	    // Stop moving second leg, with open valve
	    // 20210506_PRA - Valve normal position changed. Without control signal "#Y9_VijaStop_DesZad" is outside (helix stopped), With control signal "#Y9_VijaStop_DesZad" is inside (helix not stopped)
	    // IF #RightLegIndex=1 OR #RightLegIndex=2 THEN
	    IF #RightLegIndex=0 AND "dbTimers".Num[#i2].TT THEN
	      #Y9_VijaStop_DesZad.AutoON := True;
	    END_IF;
	    // Prepare front position for centring
	    IF "dbDigitalSensors".FOTOCELICA_VIJACENJE_DESNOSPREDAJ.InputF AND NOT #FOTOCELICA_DESNO_SPREDAJ_LATCH THEN
	      #RightLegsArrayIndex[1] := "dbDigitalSensors".FOTOCELICA_VIJACENJE_DESNOSPREDAJ.InputF;  // Reset, ko je vijacenje koncano
	      #FOTOCELICA_DESNO_SPREDAJ_LATCH := True;
	    END_IF;
	    IF #RightLegsArrayIndex[1] AND #InsertNewButtom=0 AND #MoveUPDOWN_DESNOSpredaj THEN
	      #Y11_Centri_DesSpr.AutoON := TRUE;
	    END_IF;
	    // Prepare rear position for centring
	    IF "dbDigitalSensors".FOTOCELICA_VIJACENJE_DESNOZADAJ.InputF AND NOT #FOTOCELICA_DESNO_ZADAJ_LATCH THEN
	      #RightLegsArrayIndex[2] := "dbDigitalSensors".FOTOCELICA_VIJACENJE_DESNOZADAJ.InputF;  // Reset, ko je vijacenje koncano
	      #FOTOCELICA_DESNO_ZADAJ_LATCH := True;
	    END_IF;
	    IF #RightLegsArrayIndex[2] AND #InsertNewButtom=0 AND #MoveUPDOWN_DESNOZadaj THEN
	      #Y10_Centri_DesZad.AutoON := TRUE;
	    END_IF;
	    IF #LeftLegIndex=0 OR #RightLegIndex=0 THEN
	      "dbHMIUser".CurrMachineStep := 'Transport nogic na pozicijo centriranja';
	    END_IF;
	    IF #LeftLegIndex=2 OR #RightLegIndex=2 THEN
	      "dbHMIUser".CurrMachineStep := 'Vstavi dno';
	    END_IF;
	    // **************** END - Stop ZADAJ and centring **************** //  
	    END_REGION CENTRIRANJE
	
	    // *************************************************************************** //  
	    // ************************* BEGIN - Button fastening ************************ // 
	    // *************************************************************************** // 
	    IF ("dbDigitalSensors".INDUKTIVEC_PRAVILNA_VLOZITEV_DNA_1.InputF AND "dbDigitalSensors".INDUKTIVEC_PRAVILNA_VLOZITEV_DNA_2.InputF) AND
	      #LeftLegsArrayIndex[1] AND #LeftLegsArrayIndex[2] AND #RightLegsArrayIndex[1] AND #RightLegsArrayIndex[2]
	      AND (#LeftLegIndex=2 AND #RightLegIndex=2) THEN
	      "dbTimers".Num[#i10].PRE  := #DlyToStartButtomFasten;
	      #ButtomFasting_Activated := True;
	    END_IF;
	    // *************************************************************************** // 
	    // ************************** END - Button fastening ************************* // 
	    // *************************************************************************** // 
	  
	    // *************************************************************************** //  
	    // *************** BEGIN - Start moving UP/DOWN and with helix *************** // 
	    // *************************************************************************** //
	    IF (NOT #RegimeHelix AND ("dbDigitalSensors".START_LEVO_NA_VPENJANJU.OSR OR "dbDigitalSensors".START_DESNO_NA_VPENJANJU.OSR) AND
	      (#InsertNewButtom=0 OR #InsertNewButtom=2))
	      THEN
	      #DetectStartButtom := TRUE;
	      #InsertNewButtom := 0; // Actived centering
	    ELSIF (#RegimeHelix AND (#InsertNewButtom=0 OR #InsertNewButtom=3)) THEN // Buttom removed, new inserted THEN
	      #DetectStartButtom := TRUE;
	      #InsertNewButtom := 0; // Actived centering
	    END_IF;
	
	    "dbTimers".Num[#i10].EE := (#ButtomFasting_Activated AND "dbDigitalSensors".FOTO_ZAVESA_KANAL_1.InputF AND "dbDigitalSensors".FOTO_ZAVESA_KANAL_2.InputF) 
	                               AND
	                               (
	                                #DetectStartButtom
	                               );
	
	    IF #ButtomFasting_Activated AND ("dbTimers".Num[#i10].EE AND "dbTimers".Num[#i10].DN) THEN
	      #Helix_Activated := True;
	    END_IF;    
	    IF #Helix_Activated THEN
	      #Y16_VpenjanjeDna.AutoON := True;
	      #VpenjanjeDnaActived     := True;
	      "dbHMIUser".CurrMachineStep := 'Vpenjanje dna aktivirano';
	    END_IF;
	
	    // V13_VijaLevZad_Dvig, V16_VijaLevSpr_Dvig, V6_VijaDesZad_Dvig, V9_VijaDesSpr_Dvig
	    IF #Helix_Activated THEN
	      IF NOT #MovingUPDOWN_Activated THEN // Timer expired only once
	        "dbTimers".Num[#i1].EE  := True;
	        "dbTimers".Num[#i1].PRE := #DlyToFinishButtonFasten; // 2 s
	        // PRA_20212604 - Activated #Y16_VpenjanjeDna after user press START button, before legs automatically were positioned
	        // #MovingUPDOWN_Activated := ("dbTimers".Num[#i1].EE AND "dbTimers".Num[#i1].DN) AND ("dbDigitalSensors".START_LEVO_NA_VPENJANJU.OSR OR "dbDigitalSensors".START_DESNO_NA_VPENJANJU.OSR);
	        
	        IF "dbTimers".Num[#i1].EE AND "dbTimers".Num[#i1].DN THEN
	          #MovingUPDOWN_Activated := True;
	          "dbTimers".Num[#i1].EE := FALSE;
	          "dbTimers".Num[#i1].DN := FALSE;
	        END_IF;
	      END_IF;
	  
	      IF #MovingUPDOWN_Activated AND ("dbDigitalSensors".INDUKTIVEC_PRAVILNA_VLOZITEV_DNA_1.InputF AND "dbDigitalSensors".INDUKTIVEC_PRAVILNA_VLOZITEV_DNA_2.InputF) THEN
	        "dbHMIUser".CurrMachineStep := 'Vijacenje dna v teku';
	
	        REGION VIJACENJE LEVO SPREDAJ
	        // ***** BEGIN - LEVO SPREDAJ ***** //
	        // Latch present leg
	        IF #LeftLegsArrayIndex[1] AND NOT #MoveUPDOWN_LevoSpredaj THEN
	          "dbTimers".Num[#i1].ACC := 0;
	          "dbTimers".Num[#i1].DN  := FALSE;
	          #MoveUPDOWN_LevoSpredaj := True;
	        END_IF;
	        // Start moving with present leg
	        IF #MoveUPDOWN_LevoSpredaj THEN
	          IF #LeftLegsArrayIndex[1] AND NOT #WaitLevoSpredaj THEN
	            #Y5_VijaLevSpr_Dvig.AutoON   := True;
	            #M2_SPREDAJ_LEVO.AutoON      := True;
	            #M2_SPREDAJ_LEVO.Speed1Out   := True;
	          END_IF;
	
	          IF NOT #WaitLevoSpredaj THEN
	            IF #M2_SPREDAJ_LEVO.AutoON THEN
	              "dbTimers".Num[#i1].EE  := #M2_SPREDAJ_LEVO.AutoON;
	              "dbTimers".Num[#i1].PRE  := #DlyToRotateOpposite; // 3 s
	            END_IF;
	            IF ("dbTimers".Num[#i1].EE AND NOT "dbTimers".Num[#i1].DN) THEN
	              #M2_SPREDAJ_LEVO.DirectionReq := True; // Rotate opposite for proper landing leg to button hole
	            ELSIF ("dbTimers".Num[#i1].EE AND "dbTimers".Num[#i1].DN) THEN // Leg needs to touch button and delay expired
	              #M2_SPREDAJ_LEVO.DirectionReq := False; // Change direction to start helix
	            END_IF;
	
	            // Leg hegix succeeded, wait to reach end cilinder position "DVIG_DOL=1"
	            IF (NOT #M2_SPREDAJ_LEVO.DirectionReq AND "dbTimers".Num[#i1].EE AND "dbTimers".Num[#i1].DN) AND ("IND_VIJAC_LEVO_NAPREJ" OR "dbDigitalSensors".KONCNA_POZICIJA_VIJACENJA_LEVO_NAPREJ.InputF) THEN
	              #M2_SPREDAJ_LEVO.AutoON       := False;
	              "dbTimers".Num[#i1].EE        := False;
	              "dbTimers".Num[#i1].DN        := False;
	              "dbTimers".Num[#i1].ACC       := 0;
	             
	              #WaitLevoSpredaj              := True;
	            END_IF;
	          END_IF;
	
	          // Start moving down after timer expired
	          IF #WaitLevoSpredaj THEN
	            "dbTimers".Num[#i1].EE  := True;
	            "dbTimers".Num[#i1].PRE  := #WaitTimeBeforeMoveDown;
	
	            IF "dbTimers".Num[#i1].EE AND NOT "dbTimers".Num[#i1].DN THEN
	              #Y5_VijaLevSpr_Dvig.AutoON    := True; // Dvig gor, till timer expired
	            END_IF;
	
	            // Wait to reached end position
	            IF "dbDigitalSensors".MESTO_VIJACENJE_LEVO_SPRED_DVIG_DOL.InputF THEN
	              #LeftLegsArrayIndex[1]  := "dbDigitalSensors".FOTOCELICA_VIJACENJE_LEVO_SPREDAJ.InputF; // Check if helix present at the end of moving motor down
	              #WaitLevoSpredaj        := False;
	              #MoveUPDOWN_LevoSpredaj := False;
	              #EndLevoSpredaj := True;
	            END_IF;
	          END_IF;
	        END_IF;
	        // ***** END - LEVO SPREDAJ ***** //
	        END_REGION VIJACENJE LEVO SPREDAJ
	
	        REGION VIJACENJE LEVO ZADAJ
	        // ***** BEGIN - LEVO ZADAJ ***** //
	        // Latch present leg
	        IF #LeftLegsArrayIndex[2] AND NOT #MoveUPDOWN_LevoZadaj THEN
	          "dbTimers".Num[#i2].ACC   := 0;
	          "dbTimers".Num[#i2].DN  := FALSE;
	          #MoveUPDOWN_LevoZadaj := True;
	        END_IF;
	        // Start moving with present leg
	        IF #MoveUPDOWN_LevoZadaj THEN
	          IF #LeftLegsArrayIndex[2] AND NOT #WaitLevoZadaj THEN
	            #Y4_VijaLevZad_Dvig.AutoON   := True;
	            #M1_ZADAJ_LEVO.AutoON      := True;
	            #M1_ZADAJ_LEVO.Speed1Out   := True;
	          END_IF;
	
	          IF NOT #WaitLevoZadaj THEN
	            IF #M1_ZADAJ_LEVO.AutoON THEN
	              "dbTimers".Num[#i2].EE  := #M1_ZADAJ_LEVO.AutoON;
	              "dbTimers".Num[#i2].PRE  := #DlyToRotateOpposite; // 3 s
	            END_IF;
	            IF ("dbTimers".Num[#i2].EE AND NOT "dbTimers".Num[#i2].DN) THEN
	              #M1_ZADAJ_LEVO.DirectionReq := True; // Rotate opposite for proper landing leg to button hole
	            ELSIF("dbTimers".Num[#i2].EE AND "dbTimers".Num[#i2].DN) THEN // Leg needs to touch button and delay expired
	              #M1_ZADAJ_LEVO.DirectionReq := False; // Change direction to start helix
	            END_IF;
	
	            // Leg hegix succeeded, wait to reach end cilinder position "DVIG_DOL=1"
	            IF (NOT #M1_ZADAJ_LEVO.DirectionReq AND "dbTimers".Num[#i2].EE AND "dbTimers".Num[#i2].DN) AND ("IND_VIJAC_LEVO_NAZAJ" OR "dbDigitalSensors".KONCNA_POZICIJA_VIJACENJA_LEVO_NAZAJ.InputF ) THEN
	              #M1_ZADAJ_LEVO.AutoON       := False;
	              "dbTimers".Num[#i2].EE        := False;
	              "dbTimers".Num[#i2].DN        := False;
	              "dbTimers".Num[#i2].ACC       := 0;
	
	              #WaitLevoZadaj              := True;
	            END_IF;
	          END_IF;
	
	          // Start moving down after timer expired
	          IF #WaitLevoZadaj THEN
	            "dbTimers".Num[#i2].EE  := True;
	            "dbTimers".Num[#i2].PRE  := #WaitTimeBeforeMoveDown;
	
	            IF "dbTimers".Num[#i2].EE AND NOT "dbTimers".Num[#i2].DN THEN
	              #Y4_VijaLevZad_Dvig.AutoON    := True; // Dvig gor, till timer expired
	            END_IF;
	
	            // Wait to reached end position
	            IF "dbDigitalSensors".MESTO_VIJACENJE_LEVO_ZAD_DVIG_DOL.InputF THEN
	              #LeftLegsArrayIndex[2] := "dbDigitalSensors".FOTOCELICA_VIJACENJE_LEVO_ZADAJ.InputF; // // Check if helix present at the end of moving motor down
	              #WaitLevoZadaj         := False;
	              #MoveUPDOWN_LevoZadaj  := False;
	              #EndLevoZadaj := True;
	            END_IF;
	          END_IF;
	        END_IF;
	        // ***** END - LEVO ZADAJ ***** //
	        END_REGION VIJACENJE LEVO ZADAJ
	
	        REGION VIJACENJE DESNO SPREDAJ
	        // ***** BEGIN - DESNO SPREDAJ ***** //
	        // Latch present leg
	        IF #RightLegsArrayIndex[1] AND NOT #MoveUPDOWN_DESNOSpredaj THEN
	          "dbTimers".Num[#i3].ACC   := 0;
	          "dbTimers".Num[#i3].DN  := FALSE;
	          #MoveUPDOWN_DESNOSpredaj := True;
	        END_IF;
	        // Start moving with present leg
	        IF #MoveUPDOWN_DESNOSpredaj THEN
	          IF #RightLegsArrayIndex[1] AND NOT #WaitDesnoSpredaj THEN
	            #Y3_VijaDesSpr_Dvig.AutoON   := True;
	            #M2_SPREDAJ_DESNO.AutoON      := True;
	            #M2_SPREDAJ_DESNO.Speed1Out   := True;
	          END_IF;
	
	          IF NOT #WaitDesnoSpredaj THEN
	            IF #M2_SPREDAJ_DESNO.AutoON THEN
	              "dbTimers".Num[#i3].EE  := #M2_SPREDAJ_DESNO.AutoON;
	              "dbTimers".Num[#i3].PRE  := #DlyToRotateOpposite; // 3 s
	            END_IF;
	            IF ("dbTimers".Num[#i3].EE AND NOT "dbTimers".Num[#i3].DN) THEN
	              #M2_SPREDAJ_DESNO.DirectionReq := True; // Rotate opposite for proper landing leg to button hole
	            ELSIF ("dbTimers".Num[#i3].EE AND "dbTimers".Num[#i3].DN) THEN // Leg needs to touch button and delay expir
	              #M2_SPREDAJ_DESNO.DirectionReq := False; // Change direction to start helix
	            END_IF;
	
	            // Leg hegix succeeded, wait to reach end cilinder position "DVIG_DOL=1"
	            IF (NOT #M2_SPREDAJ_DESNO.DirectionReq AND "dbTimers".Num[#i3].EE AND "dbTimers".Num[#i3].DN) AND ("IND_VIJAC_DES_NAPREJ" OR "dbDigitalSensors".KONCNA_POZICIJA_VIJACENJA_DES_NAPREJ.InputF) THEN
	              #M2_SPREDAJ_DESNO.AutoON      := False;          
	              "dbTimers".Num[#i3].EE        := False;
	              "dbTimers".Num[#i3].DN        := False;
	              "dbTimers".Num[#i3].ACC       := 0;
	
	              #WaitDesnoSpredaj             := True;
	            END_IF;
	          END_IF;
	
	          // Start moving down after timer expired
	          IF #WaitDesnoSpredaj THEN
	            "dbTimers".Num[#i3].EE  := True;
	            "dbTimers".Num[#i3].PRE  := #WaitTimeBeforeMoveDown;
	
	            IF "dbTimers".Num[#i3].EE AND NOT "dbTimers".Num[#i3].DN THEN
	              #Y3_VijaDesSpr_Dvig.AutoON    := True; // Dvig gor, till timer expired
	            END_IF;
	
	            // Wait to reached end position
	            IF "dbDigitalSensors".MESTO_VIJACENJE_DESNO_SPRED_DVIG_DOL.InputF THEN
	              #RightLegsArrayIndex[1]  := "dbDigitalSensors".FOTOCELICA_VIJACENJE_DESNOSPREDAJ.InputF; // // Check if helix present at the end of moving motor down
	              #WaitDesnoSpredaj        := False;
	              #MoveUPDOWN_DESNOSpredaj := False;
	              #EndDesnoSpredaj := True;
	            END_IF;
	          END_IF;
	        END_IF;
	        // ***** END - DESNO SPREDAJ ***** //
	        END_REGION VIJACENJE DESNO SPREDAJ
	
	        REGION VIJACENJE DESNO ZADAJ
	        // ***** BEGIN - DESNO ZADAJ ***** //
	        // Latch present leg
	        IF #RightLegsArrayIndex[2] AND NOT #MoveUPDOWN_DESNOZadaj THEN
	          "dbTimers".Num[#i4].ACC  := 0;
	          "dbTimers".Num[#i4].DN  := FALSE;
	          #MoveUPDOWN_DESNOZadaj := True;
	        END_IF;
	        // Start moving with present leg
	        IF #MoveUPDOWN_DESNOZadaj THEN
	          IF #RightLegsArrayIndex[2] AND NOT #WaitDesnoZadaj THEN
	            #Y2_VijaDesZad_Dvig.AutoON   := True;
	            #M1_ZADAJ_DESNO.AutoON      := True;
	            #M1_ZADAJ_DESNO.Speed1Out   := True;
	          END_IF;
	
	          IF NOT #WaitDesnoZadaj THEN
	            IF #M1_ZADAJ_DESNO.AutoON THEN
	              "dbTimers".Num[#i4].EE  := #M1_ZADAJ_DESNO.AutoON;
	              "dbTimers".Num[#i4].PRE  := #DlyToRotateOpposite; // 3 s
	            END_IF;
	            IF ("dbTimers".Num[#i4].EE AND NOT "dbTimers".Num[#i4].DN) THEN
	              #M1_ZADAJ_DESNO.DirectionReq := True; // Rotate opposite for proper landing leg to button hole
	            ELSIF ("dbTimers".Num[#i4].EE AND "dbTimers".Num[#i4].DN) THEN // // Leg needs to touch button and delay expired
	              #M1_ZADAJ_DESNO.DirectionReq := False; // Change direction to start helix
	            END_IF;
	
	            // Leg hegix succeeded, wait to reach end cilinder position "DVIG_DOL=1"
	            IF (NOT #M1_ZADAJ_DESNO.DirectionReq AND "dbTimers".Num[#i4].EE AND "dbTimers".Num[#i4].DN) AND ("IND_VIJAC_DES_NAZAJ" OR "dbDigitalSensors".KONCNA_POZICIJA_VIJACENJA_DES_NAZAJ.InputF) THEN 
	              #M1_ZADAJ_DESNO.AutoON       := False;
	              "dbTimers".Num[#i4].EE       := False;
	              "dbTimers".Num[#i4].DN       := False;
	              "dbTimers".Num[#i4].ACC      := 0;
	
	              #WaitDesnoZadaj              := True;
	            END_IF;
	          END_IF;
	
	          // Start moving down after timer expired
	          IF #WaitDesnoZadaj THEN
	            "dbTimers".Num[#i4].EE  := True;
	            "dbTimers".Num[#i4].PRE  := #WaitTimeBeforeMoveDown;
	
	            IF "dbTimers".Num[#i4].EE AND NOT "dbTimers".Num[#i4].DN THEN
	              #Y2_VijaDesZad_Dvig.AutoON    := True; // Dvig gor, till timer expired
	            END_IF;
	
	            // Wait to reached end position
	            IF "dbDigitalSensors".MESTO_VIJACENJE_DESNO_ZAD_DVIG_DOL.InputF THEN
	              #RightLegsArrayIndex[2] := "dbDigitalSensors".FOTOCELICA_VIJACENJE_DESNOZADAJ.InputF; // // Check if helix present at the end of moving motor down
	              #WaitDesnoZadaj        := False;
	              #MoveUPDOWN_DESNOZadaj := False;
	              #EndDesnoZadaj := True;
	            END_IF;
	          END_IF;
	        END_IF;
	        // ***** END - DESNO ZADAJ ***** //
	        END_REGION VIJACENJE DESNO ZADAJ
	
	        // Next step
	        IF (#EndLevoSpredaj AND #EndLevoZadaj AND #EndDesnoSpredaj AND #EndDesnoZadaj) AND
	           ("dbDigitalSensors".FOTO_ZAVESA_KANAL_1.InputF AND "dbDigitalSensors".FOTO_ZAVESA_KANAL_2.InputF)     
	          THEN
	          "dbTimers".Num[#i1].EE  := False;
	          "dbTimers".Num[#i1].DN  := False;
	          "dbTimers".Num[#i1].ACC := 0;
	          "dbTimers".Num[#i2].EE  := False;
	          "dbTimers".Num[#i2].DN  := False;
	          "dbTimers".Num[#i2].ACC := 0;
	          "dbTimers".Num[#i3].EE  := False;
	          "dbTimers".Num[#i3].DN  := False;
	          "dbTimers".Num[#i3].ACC := 0;
	          "dbTimers".Num[#i4].EE  := False;
	          "dbTimers".Num[#i4].DN  := False;
	          "dbTimers".Num[#i4].ACC := 0;
	          "dbTimers".Num[#i10].EE  := False;
	          "dbTimers".Num[#i10].DN  := False;
	          "dbTimers".Num[#i10].ACC := 0;
	          #TotalButtomPlateCounter := #TotalButtomPlateCounter + 1;
	
	          #CurrentStep := 20;
	        END_IF;
	  
	      END_IF; // #MovingUPDOWN_ready
	    END_IF;   // #Helix_Activated
	    // *************************************************************************** // 
	    // *************** END - Start moving UP/DOWN and with helix ***************** //
	    // *************************************************************************** // 
	
	  20:  // Remove button plate - wait user to remove button plate
	  "dbHMIUser".CurrMachineStep := 'Odstrani dno iz naprave';
	  #MovingUPDOWN_Activated := False; // 20210426_PRA Added to reset before plate is removed. Used in fcUtilities->timer: StandbyTimeTrakaVijac
	  #InsertNewButtom := 1;
	
	  IF #LeftLegsArrayIndex[1] OR #LeftLegsArrayIndex[2] THEN
	    #LeftLegIndex  := 2; // vijačenje neuspešno, ponovi vijačenje z istimi nogicami
	  ELSE
	    #LeftLegIndex  := 0; // vijačenje uspešno
	  END_IF;
	  IF #RightLegsArrayIndex[1] OR #RightLegsArrayIndex[2] THEN
	    #RightLegIndex := 2; // vijačenje neuspešno, ponovi vijačenje z istimi nogicami
	  ELSE
	    #RightLegIndex := 0; // vijačenje uspešno
	  END_IF;
	
	  IF #LeftLegIndex=0 AND #RightLegIndex=0 THEN
	    #LegsReadyOnPosToHelix := False;
	  END_IF;
	
	  REGION CENTRIRANJE AT END
	  // *************** BEGIN - Stop ZADAJ and centring *************** //
	  (* // 20210506_PRA In normal position #Y13_VijaStop_LevZad is outside
	  IF #LeftLegIndex=1 OR #LeftLegIndex=2 THEN
	    #Y13_VijaStop_LevZad.AutoON := True;  // Stop moving second leg, with open valve
	  END_IF;
	  *)
	  IF #LeftLegsArrayIndex[1] THEN
	    #Y15_Centri_LevSpr.AutoON := TRUE;
	  END_IF;
	  IF #LeftLegsArrayIndex[2] THEN
	    #Y14_Centri_LevZad.AutoON := TRUE;
	  END_IF;
	
	  (* // 20210506_PRA In normal position #Y9_VijaStop_DesZad is outside
	  IF #RightLegIndex=1 OR #RightLegIndex=2 THEN
	    #Y9_VijaStop_DesZad.AutoON := True; // Stop moving second leg, with open valve
	  END_IF;
	  *)
	  IF #RightLegsArrayIndex[1] THEN
	    #Y11_Centri_DesSpr.AutoON := TRUE;
	  END_IF;
	  IF #RightLegsArrayIndex[2] THEN
	    #Y10_Centri_DesZad.AutoON := TRUE;
	  END_IF;
	  // **************** END - Stop ZADAJ and centring **************** //  
	  END_REGION CENTRIRANJE
	
	  "dbTimers".Num[#i1].FR    := False;
	  "dbTimers".Num[#i2].FR    := False;
	  "dbTimers".Num[#i3].FR    := False;
	  "dbTimers".Num[#i4].FR    := False;
	
	  "dbTimers".Num[#i1].EE := ("dbDigitalSensors".FOTO_ZAVESA_KANAL_1.InputF AND "dbDigitalSensors".FOTO_ZAVESA_KANAL_2.InputF) AND
	                            "dbDigitalSensors".MESTO_VIJACENJE_LEVO_SPRED_DVIG_DOL.InputF AND "dbDigitalSensors".MESTO_VIJACENJE_LEVO_SPRED_DVIG_DOL.InputF AND
	                            "dbDigitalSensors".MESTO_VIJACENJE_DESNO_SPRED_DVIG_DOL.InputF AND "dbDigitalSensors".MESTO_VIJACENJE_DESNO_SPRED_DVIG_DOL.InputF;
	                            // 20210429_PRA Start next legs positions even if buttom was not removed from machine and buttom AND still present
	                            // (NOT "dbDigitalSensors".INDUKTIVEC_PRAVILNA_VLOZITEV_DNA_1.InputF AND NOT "dbDigitalSensors".INDUKTIVEC_PRAVILNA_VLOZITEV_DNA_2.InputF)
	  "dbTimers".Num[#i1].PRE := #WEndTimeToRemovePlate;
	  IF "dbTimers".Num[#i1].EE AND "dbTimers".Num[#i1].DN THEN
	    // *************** BEGIN - Preveri ali so bile nogice zvijacene *************** //
	    #LeftLegsArrayIndex[1] := "dbDigitalSensors".FOTOCELICA_VIJACENJE_LEVO_SPREDAJ.InputF;
	    #LeftLegsArrayIndex[2] := "dbDigitalSensors".FOTOCELICA_VIJACENJE_LEVO_ZADAJ.InputF;
	    #RightLegsArrayIndex[1] := "dbDigitalSensors".FOTOCELICA_VIJACENJE_DESNOSPREDAJ.InputF;
	    #RightLegsArrayIndex[2] := "dbDigitalSensors".FOTOCELICA_VIJACENJE_DESNOZADAJ.InputF;
	    // **************** END - Preveri ali so bile nogice zvijacene **************** //  
	    #CurrentStep := 21;
	  END_IF;
	  
	  21:  // Jump to initial step
	  "dbTimers".Num[#i1].EE  := False;
	  "dbTimers".Num[#i1].DN  := False;
	
	  #InitPosition := False;
	  #CurrentStep := 1; // Check conditions on init step
	
	END_CASE;
	
	// ALARMS SECTION
	  // Alarm 1
	  IF #Y8_VijaLocev_Des.Alarm THEN
	    "dbAlarms".PLI[#PLIIndex, 1] := 1;
	  END_IF;
	  
	  // Alarm 2
	  IF #Y9_VijaStop_DesZad.Alarm THEN
	    "dbAlarms".PLI[#PLIIndex, 2] := 1;
	  END_IF;
	  
	  // Alarm 3
	  IF #Y2_VijaDesZad_Dvig.Alarm THEN
	    "dbAlarms".PLI[#PLIIndex, 3] := 1;
	  END_IF;
	  
	  // Alarm 4
	  IF #Y10_Centri_DesZad.Alarm THEN
	    "dbAlarms".PLI[#PLIIndex, 4] := 1;
	  END_IF;
	  
	  // Alarm 5
	  IF #Y3_VijaDesSpr_Dvig.Alarm THEN
	    "dbAlarms".PLI[#PLIIndex, 5] := 1;
	  END_IF;
	
	  // Alarm 6
	  IF #Y11_Centri_DesSpr.Alarm THEN
	    "dbAlarms".PLI[#PLIIndex, 6] := 1;
	  END_IF;
	
	  // Alarm 7
	  IF #Y12_VijaLocev_Lev.Alarm THEN 
	    "dbAlarms".PLI[#PLIIndex, 7] := 1;
	  END_IF;
	  
	  // Alarm 8
	  IF #Y13_VijaStop_LevZad.Alarm THEN 
	    "dbAlarms".PLI[#PLIIndex, 8] := 1;
	  END_IF;
	  
	  // Alarm 9
	  IF #Y4_VijaLevZad_Dvig.Alarm THEN
	    "dbAlarms".PLI[#PLIIndex, 9] := 1;
	  END_IF;
	  
	  // Alarm 10
	  IF #Y14_Centri_LevZad.Alarm THEN
	    "dbAlarms".PLI[#PLIIndex, 10] := 1;
	  END_IF;
	  
	  // Alarm 11
	  IF #Y5_VijaLevSpr_Dvig.Alarm THEN
	    "dbAlarms".PLI[#PLIIndex, 11] := 1;
	  END_IF;
	  
	  // Alarm 12
	  IF #Y15_Centri_LevSpr.Alarm THEN
	    "dbAlarms".PLI[#PLIIndex, 12] := 1;
	  END_IF;
	
	  // Alarm 13
	  IF #Y16_VpenjanjeDna.Alarm THEN
	    "dbAlarms".PLI[#PLIIndex, 13] := 1;
	  END_IF;
	
	  // Alarm 14
	  IF #M1_ZADAJ_LEVO.Alarm THEN
	    "dbAlarms".PLI[#PLIIndex, 14] := 1;
	  END_IF;
	
	  // Alarm 15
	  IF #M2_SPREDAJ_LEVO.Alarm THEN
	    "dbAlarms".PLI[#PLIIndex, 15] := 1;
	  END_IF;
	
	  // Alarm 16
	  IF #M1_ZADAJ_DESNO.Alarm THEN
	    "dbAlarms".PLI[#PLIIndex, 16] := 1;
	  END_IF;
	
	  // Alarm 17
	  IF #M2_SPREDAJ_DESNO.Alarm THEN
	    "dbAlarms".PLI[#PLIIndex, 17] := 1;
	  END_IF;
	
	  // Alarm 18
	  IF #VKLOP_M_TRAKA_VIJACNIKA.Alarm THEN
	    "dbAlarms".PLI[#PLIIndex, 18] := 1;
	  END_IF;
	
	  // Alarm 19
	  // Začetne pozicije vijačnega dela niso dosežene
	  IF #CurrentStep = 1 AND #IEC_TimerOnDly_DN_1 THEN // NOT #InitPosition
	    "dbAlarms".PLI[#PLIIndex, 19] := 1;
	  END_IF;
	
	  // Alarm 20
	  // Manjka ena od nogic na pozicijah za vijačenje-ročno odstrani nogice
	  IF (#CurrentStep >= 3 AND #CurrentStep <= 5) AND
	    (#LeftLegsArrayIndex[1] XOR #LeftLegsArrayIndex[2] XOR #RightLegsArrayIndex[1] XOR #RightLegsArrayIndex[2])
	  THEN
	    "dbUnit".Unit[1].StartStop := False;
	    "dbAlarms".PLI[#PLIIndex, 20] := 1;
	  END_IF;
	
	  // Alarm 21 - Added 20210512_PRA
	  // Dovoljeni čas vijačenja nogice levo-spredaj potekel
	  "dbTimers".Num[#i5].EE := (#PhaseStatus=5 AND #CurrentStep = 10) AND #MovingUPDOWN_Activated AND #MoveUPDOWN_LevoSpredaj AND NOT #WaitLevoSpredaj;
	  "dbTimers".Num[#i5].PRE := #TimeoutToEndHelix;
	  IF "dbTimers".Num[#i5].EE AND "dbTimers".Num[#i5].DN
	  THEN
	    "dbUnit".Unit[1].StartStop := False;
	    "dbAlarms".PLI[#PLIIndex, 21] := 1;
	  END_IF;
	
	  // Alarm 22 - Added 20210512_PRA
	  // Dovoljeni čas vijačenja nogice levo-zadaj potekel
	  "dbTimers".Num[#i6].EE := (#PhaseStatus=5 AND #CurrentStep = 10) AND #MovingUPDOWN_Activated AND #MoveUPDOWN_LevoZadaj AND NOT #WaitLevoZadaj;
	  "dbTimers".Num[#i6].PRE := #TimeoutToEndHelix;
	  IF "dbTimers".Num[#i6].EE AND "dbTimers".Num[#i6].DN
	  THEN
	    "dbUnit".Unit[1].StartStop := False;
	    "dbAlarms".PLI[#PLIIndex, 22] := 1;
	  END_IF;
	
	  // Alarm 23 - Added 20210512_PRA
	  // Dovoljeni čas vijačenja nogice desno-spredaj potekel
	  "dbTimers".Num[#i7].EE := (#PhaseStatus=5 AND #CurrentStep = 10) AND #MovingUPDOWN_Activated AND #MoveUPDOWN_DESNOSpredaj AND NOT #WaitDesnoSpredaj;
	  "dbTimers".Num[#i7].PRE := #TimeoutToEndHelix;
	  IF "dbTimers".Num[#i7].EE AND "dbTimers".Num[#i7].DN
	  THEN
	    "dbUnit".Unit[1].StartStop := False;
	    "dbAlarms".PLI[#PLIIndex, 23] := 1;
	  END_IF;
	
	  // Alarm 24 - Added 20210512_PRA
	  // Dovoljeni čas vijačenja nogice desno-zadaj potekel
	  "dbTimers".Num[#i8].EE := (#PhaseStatus=5 AND #CurrentStep = 10) AND #MovingUPDOWN_Activated AND #MoveUPDOWN_DESNOZadaj AND NOT #WaitDesnoZadaj;
	  "dbTimers".Num[#i8].PRE := #TimeoutToEndHelix;
	  IF "dbTimers".Num[#i8].EE AND "dbTimers".Num[#i8].DN
	  THEN
	    "dbUnit".Unit[1].StartStop := False;
	    "dbAlarms".PLI[#PLIIndex, 24] := 1;
	  END_IF;
	
	  // Alarms in running state
	  IF #PhaseStatus = 5 THEN
	    IF (NOT #AlarmPresentOLD AND #AlarmPresent) OR (NOT #InitPositionOLD AND #InitPosition) THEN
	      ; // #CurrentStep := 6;
	    END_IF;
	  END_IF;
	
	#AlarmPresentOLD      := #AlarmPresent;
	#InitPositionOLD      := #InitPosition;
	
	IF (#CurrentStep = 10) THEN
	  #LeftLegIndexOLD      := #LeftLegIndex;
	  #RightLegIndexOLD     := #RightLegIndex;
	END_IF;
END_FUNCTION_BLOCK

FUNCTION_BLOCK "ph_LegsShifter_2"
{ S7_Optimized_Access := 'TRUE' }
VERSION : 0.1
   VAR_IN_OUT 
      Y17_RotCilipozDesno : "udtDigitalValve";
      Y18_RotCilipozLevo : "udtDigitalValve";
      Y6_DrcaLocev_Des : "udtDigitalValve";
      Y7_DrcaLocev_Lev : "udtDigitalValve";
   END_VAR

   VAR RETAIN
      CurrentStep { ExternalAccessible := 'False'; ExternalVisible := 'False'; ExternalWritable := 'False'} : Int;
      PhaseStatus { ExternalAccessible := 'False'; ExternalVisible := 'False'; ExternalWritable := 'False'} : Int;   // // 0=IDLE, 5=RUNNING, 6=HOLD
      Mode { ExternalAccessible := 'False'; ExternalVisible := 'False'; ExternalWritable := 'False'} : SInt;
      AlarmPresent { ExternalAccessible := 'False'; ExternalVisible := 'False'; ExternalWritable := 'False'} : Bool;
      InitPosition { ExternalAccessible := 'False'; ExternalVisible := 'False'; ExternalWritable := 'False'} : Bool;
   END_VAR
   VAR 
      StartCmd { ExternalAccessible := 'False'; ExternalVisible := 'False'; ExternalWritable := 'False'} : Bool;
      AlarmPresentOLD { ExternalAccessible := 'False'; ExternalVisible := 'False'; ExternalWritable := 'False'} : Bool;
      InitPositionOLD { ExternalAccessible := 'False'; ExternalVisible := 'False'; ExternalWritable := 'False'} : Bool;
      IEC_TimerOnDly_1 {InstructionName := 'TONR_TIME'; LibVersion := '1.0'; ExternalAccessible := 'False'; ExternalVisible := 'False'; ExternalWritable := 'False'; S7_SetPoint := 'False'} : TONR_TIME;
      IEC_TimerOnDly_2 {InstructionName := 'TONR_TIME'; LibVersion := '1.0'; ExternalAccessible := 'False'; ExternalVisible := 'False'; ExternalWritable := 'False'; S7_SetPoint := 'False'} : TONR_TIME;
      IEC_TimerOnDly_3 {InstructionName := 'TONR_TIME'; LibVersion := '1.0'; ExternalAccessible := 'False'; ExternalVisible := 'False'; ExternalWritable := 'False'; S7_SetPoint := 'False'} : TONR_TIME;
      IEC_TimerOnDly_4 {InstructionName := 'TONR_TIME'; LibVersion := '1.0'; ExternalAccessible := 'False'; ExternalVisible := 'False'; ExternalWritable := 'False'; S7_SetPoint := 'False'} : TONR_TIME;
      IEC_TimerOnDly_5 {InstructionName := 'TONR_TIME'; LibVersion := '1.0'; ExternalAccessible := 'False'; ExternalVisible := 'False'; ExternalWritable := 'False'; S7_SetPoint := 'False'} : TONR_TIME;
      IEC_TimerOnDly_6 {InstructionName := 'TONR_TIME'; LibVersion := '1.0'; ExternalAccessible := 'False'; ExternalVisible := 'False'; ExternalWritable := 'False'; S7_SetPoint := 'False'} : TONR_TIME;
      IEC_TimerOnDly_7 {InstructionName := 'TONR_TIME'; LibVersion := '1.0'; ExternalAccessible := 'False'; ExternalVisible := 'False'; ExternalWritable := 'False'; S7_SetPoint := 'False'} : TONR_TIME;
      IEC_TimerOnDly_8 {InstructionName := 'TONR_TIME'; LibVersion := '1.0'; ExternalAccessible := 'False'; ExternalVisible := 'False'; ExternalWritable := 'False'; S7_SetPoint := 'False'} : TONR_TIME;
      IEC_TimerOnDly_9 {InstructionName := 'TONR_TIME'; LibVersion := '1.0'; ExternalAccessible := 'False'; ExternalVisible := 'False'; ExternalWritable := 'False'; S7_SetPoint := 'False'} : TONR_TIME;
      IEC_TimerOnDly_10 {InstructionName := 'TONR_TIME'; LibVersion := '1.0'; ExternalAccessible := 'False'; ExternalVisible := 'False'; ExternalWritable := 'False'; S7_SetPoint := 'False'} : TONR_TIME;
      IEC_TimerOnDly_ET_1 { ExternalAccessible := 'False'; ExternalVisible := 'False'; ExternalWritable := 'False'} : Time;
      IEC_TimerOnDly_ET_2 { ExternalAccessible := 'False'; ExternalVisible := 'False'; ExternalWritable := 'False'} : Time;
      IEC_TimerOnDly_ET_3 { ExternalAccessible := 'False'; ExternalVisible := 'False'; ExternalWritable := 'False'} : Time;
      IEC_TimerOnDly_ET_4 { ExternalAccessible := 'False'; ExternalVisible := 'False'; ExternalWritable := 'False'} : Time;
      IEC_TimerOnDly_ET_5 { ExternalAccessible := 'False'; ExternalVisible := 'False'; ExternalWritable := 'False'} : Time;
      IEC_TimerOnDly_ET_6 { ExternalAccessible := 'False'; ExternalVisible := 'False'; ExternalWritable := 'False'} : Time;
      IEC_TimerOnDly_ET_7 { ExternalAccessible := 'False'; ExternalVisible := 'False'; ExternalWritable := 'False'} : Time;
      IEC_TimerOnDly_ET_8 { ExternalAccessible := 'False'; ExternalVisible := 'False'; ExternalWritable := 'False'} : Time;
      IEC_TimerOnDly_ET_9 { ExternalAccessible := 'False'; ExternalVisible := 'False'; ExternalWritable := 'False'} : Time;
      IEC_TimerOnDly_ET_10 { ExternalAccessible := 'False'; ExternalVisible := 'False'; ExternalWritable := 'False'} : Time;
      IEC_TimerOnDly_DN_1 { ExternalAccessible := 'False'; ExternalVisible := 'False'; ExternalWritable := 'False'} : Bool;
      IEC_TimerOnDly_DN_2 { ExternalAccessible := 'False'; ExternalVisible := 'False'; ExternalWritable := 'False'} : Bool;
      IEC_TimerOnDly_DN_3 { ExternalAccessible := 'False'; ExternalVisible := 'False'; ExternalWritable := 'False'} : Bool;
      IEC_TimerOnDly_DN_4 { ExternalAccessible := 'False'; ExternalVisible := 'False'; ExternalWritable := 'False'} : Bool;
      IEC_TimerOnDly_DN_5 { ExternalAccessible := 'False'; ExternalVisible := 'False'; ExternalWritable := 'False'} : Bool;
      IEC_TimerOnDly_DN_6 { ExternalAccessible := 'False'; ExternalVisible := 'False'; ExternalWritable := 'False'} : Bool;
      IEC_TimerOnDly_DN_7 { ExternalAccessible := 'False'; ExternalVisible := 'False'; ExternalWritable := 'False'} : Bool;
      IEC_TimerOnDly_DN_8 { ExternalAccessible := 'False'; ExternalVisible := 'False'; ExternalWritable := 'False'} : Bool;
      IEC_TimerOnDly_DN_9 { ExternalAccessible := 'False'; ExternalVisible := 'False'; ExternalWritable := 'False'} : Bool;
      IEC_TimerOnDly_DN_10 { ExternalAccessible := 'False'; ExternalVisible := 'False'; ExternalWritable := 'False'} : Bool;
      FillingLineSelector { ExternalAccessible := 'False'; ExternalVisible := 'False'; ExternalWritable := 'False'} : USInt;
      InletLineStep { ExternalAccessible := 'False'; ExternalVisible := 'False'; ExternalWritable := 'False'} : SInt;
      LeftOutletLineStep { ExternalAccessible := 'False'; ExternalVisible := 'False'; ExternalWritable := 'False'} : SInt;
      RightOutletLineStep { ExternalAccessible := 'False'; ExternalVisible := 'False'; ExternalWritable := 'False'} : SInt;
   END_VAR
   VAR RETAIN
      TimeToLoadInletLine { S7_SetPoint := 'True'} : Int := 20;
      TimeToReleaseInletLine { S7_SetPoint := 'True'} : Int := 10;
      TimeToReleaseOutletLine { S7_SetPoint := 'True'} : Int := 10;
   END_VAR
   VAR 
      LeftLegIndex { ExternalAccessible := 'False'; ExternalVisible := 'False'; ExternalWritable := 'False'} : SInt;
      RightLegIndex { ExternalAccessible := 'False'; ExternalVisible := 'False'; ExternalWritable := 'False'} : SInt;
      LeftFirstLegIndex { ExternalAccessible := 'False'; ExternalVisible := 'False'; ExternalWritable := 'False'} : SInt;
      RightFirstLegIndex { ExternalAccessible := 'False'; ExternalVisible := 'False'; ExternalWritable := 'False'} : SInt;
      DRCA_DESNO_LATCH { ExternalAccessible := 'False'; ExternalVisible := 'False'; ExternalWritable := 'False'} : Bool;
      DRCA_LEVO_LATCH { ExternalAccessible := 'False'; ExternalVisible := 'False'; ExternalWritable := 'False'} : Bool;
   END_VAR

   VAR_TEMP 
      i : Int;
      i1 : Int;
      i2 : Int;
      i3 : Int;
      i4 : Int;
      i5 : Int;
      i6 : Int;
      i7 : Int;
      i8 : Int;
      i9 : Int;
      i10 : Int;
   END_VAR

   VAR CONSTANT 
      ReleaseValOnBeltSepaTime : Int := 20;
      PLIIndex : Int := 2;
   END_VAR


BEGIN
	#i1   := #PLIIndex;                          // 1
	#i2   := #PLIIndex + "MaxPLITimersIndex";    // 5
	#i3   := #PLIIndex + 2*"MaxPLITimersIndex";  // 9
	#i4   := #PLIIndex + 3*"MaxPLITimersIndex";  // 13
	#i5   := #PLIIndex + 4*"MaxPLITimersIndex";  // 17
	#i6   := #PLIIndex + 5*"MaxPLITimersIndex";  // 21
	#i7   := #PLIIndex + 6*"MaxPLITimersIndex";  // 25
	#i8   := #PLIIndex + 7*"MaxPLITimersIndex";  // 29
	#i9   := #PLIIndex + 8*"MaxPLITimersIndex";  // 33
	#i10  := #PLIIndex + 9*"MaxPLITimersIndex";  // 37
	
	// Check alarms
	#AlarmPresent := 0;
	FOR #i := 1 TO 32 DO
	  IF "dbAlarms".PLI[#PLIIndex, #i] THEN
	    #AlarmPresent := 1;
	    // #StartCmd     := False;
	  END_IF;
	  IF "AlarmAck" THEN
	    "dbAlarms".PLI[#PLIIndex, #i] := 0;
	  END_IF;
	END_FOR;
	
	// Timers section
	#IEC_TimerOnDly_DN_1 := 0;
	#IEC_TimerOnDly_1(IN := #CurrentStep = 2 AND NOT #InitPosition,
	                  R := #CurrentStep <> 2,
	                  PT := T#3s,
	                  Q => #IEC_TimerOnDly_DN_1,
	                  ET => #IEC_TimerOnDly_ET_1);
	
	// PHASE STATUS
	#PhaseStatus := 0;
	IF #CurrentStep >= 1 AND #StartCmd THEN
	  #PhaseStatus := 5;
	END_IF;
	IF #CurrentStep >= 1 AND NOT #StartCmd THEN
	  #PhaseStatus := 7;
	END_IF;
	IF #CurrentStep >= 1 AND #AlarmPresent THEN
	  #PhaseStatus := 6;
	END_IF;
	
	// Stop phase if START CMD=0
	IF NOT #StartCmd AND #CurrentStep > 0 THEN
	  #CurrentStep := 0;
	END_IF;
	
	CASE #CurrentStep OF
	  0: // Sequence permissives
	  IF (#StartCmd AND TRUE) THEN // Local  mode
	    IF #PhaseStatus=0 THEN
	      #CurrentStep := 2;
	    END_IF;
	    
	    #InitPosition := False;
	  END_IF;
	
	  2: // Check initial positions
	    #InitPosition := ("dbDigitalSensors".ROTACIJSKI_CIL_SREDINA.InputF AND "dbDigitalSensors".LOC_DRCA_LEVO_NAPREJ.InputF AND "dbDigitalSensors".LOC_DRCA_DESNO_NAPREJ.InputF);
	
	    IF #InitPosition AND NOT "dbUnit".Unit[1].AlarmsPresent THEN
	      #CurrentStep := 3;
	    END_IF;
	
	  3: // Check initial positions
	    #LeftLegIndex        := 0; // Reset št. nogic izpusta iz drce. Do NOT reset when step change 10->20
	    #RightLegIndex       := 0; // Reset št. nogic izpusta iz drce. Do NOT reset when step change 10->20
	
	    #LeftFirstLegIndex   := 0;
	    #RightFirstLegIndex  := 0;
	
	    // Preveri, če so prisotne nogice na vijacnem delu
	    IF ("dbDigitalSensors".FOTOCELICA_LOC_TRAK_LEVO1.InputF AND "dbDigitalSensors".FOTOCELICA_LOC_TRAK_LEVO2.InputF) THEN
	      #LeftLegIndex        := 2; // Nastavi št. nogic na 2
	      #LeftFirstLegIndex   := 2; // Nastavi št. nogic na 2
	    ELSIF "dbDigitalSensors".FOTOCELICA_LOC_TRAK_LEVO1.InputF THEN
	      #LeftLegIndex        := 1;
	      #LeftFirstLegIndex   := 1; // Nastavi št. nogic na 1
	    END_IF;
	    // Preveri, če so prisotne nogice na vijacnem delu
	    IF ("dbDigitalSensors".FOTOCELICA_LOC_TRAK_DESNO1.InputF AND "dbDigitalSensors".FOTOCELICA_LOC_TRAK_DESNO2.InputF) THEN
	       #RightLegIndex       := 2; // Nastavi št. nogic na 2
	       #RightFirstLegIndex  := 2; // Nastavi št. nogic na 2
	    ELSIF "dbDigitalSensors".FOTOCELICA_LOC_TRAK_DESNO1.InputF THEN
	      #RightLegIndex        := 1;
	      #RightFirstLegIndex   := 1; // Nastavi št. nogic na 1
	    END_IF;
	
	    #Mode := 1; // first fllling LEVO to the full then DESNO to the full
	    #CurrentStep := 5;
	
	  5: // Init variables
	    "dbTimers".Num[#i1].EE    := False;
	    "dbTimers".Num[#i2].EE    := False;
	    "dbTimers".Num[#i3].EE    := False;
	    "dbTimers".Num[#i4].EE    := False;
	    "dbTimers".Num[#i5].EE    := False;
	    "dbTimers".Num[#i6].EE    := False;
	    "dbTimers".Num[#i7].EE    := False;
	    "dbTimers".Num[#i8].EE    := False;
	    "dbTimers".Num[#i9].EE    := False;
	    "dbTimers".Num[#i10].EE   := False;
	
	    "dbTimers".Num[#i1].FR    := False;
	    "dbTimers".Num[#i2].FR    := False;
	    "dbTimers".Num[#i3].FR    := False;
	    "dbTimers".Num[#i4].FR    := False;
	    "dbTimers".Num[#i5].FR    := False;
	    "dbTimers".Num[#i6].FR    := False;
	    "dbTimers".Num[#i7].FR    := False;
	    "dbTimers".Num[#i8].FR    := False;
	    "dbTimers".Num[#i9].FR    := False;
	    "dbTimers".Num[#i10].FR   := False;
	    #DRCA_LEVO_LATCH          := False;
	    #DRCA_DESNO_LATCH         := False;
	  
	    #InletLineStep := 0;
	    #LeftOutletLineStep  := 0;
	    #RightOutletLineStep := 0;
	    #FillingLineSelector := 1;
	
	    #CurrentStep := 6;
	
	  6:// Select Mode
	    IF #Mode=1 THEN
	      #CurrentStep := 10;
	    ELSIF #Mode=2 THEN  
	      #CurrentStep := 20;
	    END_IF;
	
	  10: // Fill single line LEVO and then line DESNO till each line gets full
	    // ******************* BEGIN - ALARM STATE *********** // 
	    IF NOT #AlarmPresent THEN
	      "dbTimers".Num[#i1].FR    := False;
	      "dbTimers".Num[#i2].FR    := False;
	      "dbTimers".Num[#i3].FR    := False;
	    ELSE
	      "dbTimers".Num[#i1].FR    := True;
	      "dbTimers".Num[#i2].FR    := True;
	      "dbTimers".Num[#i3].FR    := True;
	    END_IF;
	    // ********************* END - ALARM STATE ************ // 
	
	    // Fill line LEVO
	    REGION MODE = 1 INLET HELIXS - rotation cylinder
	    // 20210506_PRA - END_IF; Check FOTOCELICA_PRED_MESTOM_LOCEVANJA only once IF "dbDigitalSensors".FOTOCELICA_PRED_MESTOM_LOCEVANJA.InputF THEN
	      IF #FillingLineSelector=1 THEN
	        // Fill line LEVO, if leg present infront of rotation cilinder
	        IF NOT "dbDigitalSensors".FOTOCELICA_VSTOP_DRCA_LEVO.InputF AND "dbDigitalSensors".FOTOCELICA_PRED_MESTOM_LOCEVANJA.InputF AND (#InletLineStep=0) THEN
	          #InletLineStep      := 1;
	          "dbTimers".Num[#i1].EE    := True;
	          "dbTimers".Num[#i1].PRE   := #TimeToLoadInletLine; // 10s
	        ELSIF (#InletLineStep =1) AND NOT "dbDigitalSensors".FOTOCELICA_VSTOP_DRCA_LEVO.InputF AND "dbTimers".Num[#i1].TT THEN
	          "dbTimers".Num[#i1].EE    := True;
	          #Y18_RotCilipozLevo.AutoON := True;
	        ELSIF "dbTimers".Num[#i1].EE AND "dbTimers".Num[#i1].DN AND (#InletLineStep =1) THEN
	          "dbTimers".Num[#i1].ACC    := 0;
	          #InletLineStep      := 2;
	        ELSIF (#InletLineStep=2) THEN
	          "dbTimers".Num[#i1].EE    := True;
	          "dbTimers".Num[#i1].PRE   := #TimeToReleaseInletLine;
	          IF ("dbTimers".Num[#i1].EE AND "dbTimers".Num[#i1].DN AND "dbTimers".Num[#i1].ACC>0) THEN
	            "dbTimers".Num[#i1].EE    := FALSE;
	            #InletLineStep      := 0;
	          END_IF;
	        END_IF;
	
	        IF "dbDigitalSensors".FOTOCELICA_VSTOP_DRCA_LEVO.InputF THEN // Go to filling opposite line, if line is full
	
	          #InletLineStep       := 3;
	          #FillingLineSelector := 2;
	        END_IF;
	
	      ELSIF #FillingLineSelector=2 THEN
	        // Fill line DESNO, if leg present infront of rotation cilinder
	        IF NOT "dbDigitalSensors".FOTOCELICA_VSTOP_DRCA_DESNO.InputF AND "dbDigitalSensors".FOTOCELICA_PRED_MESTOM_LOCEVANJA.InputF AND (#InletLineStep=3) THEN
	          #InletLineStep      := 4;
	          "dbTimers".Num[#i1].EE    := True;
	          "dbTimers".Num[#i1].PRE   := #TimeToLoadInletLine; // 10s
	        ELSIF (#InletLineStep =4) AND NOT "dbDigitalSensors".FOTOCELICA_VSTOP_DRCA_DESNO.InputF AND "dbTimers".Num[#i1].TT THEN
	          "dbTimers".Num[#i1].EE    := True;
	          #Y17_RotCilipozDesno.AutoON := True;
	        ELSIF "dbTimers".Num[#i1].EE AND "dbTimers".Num[#i1].DN AND (#InletLineStep =4) THEN
	          "dbTimers".Num[#i1].ACC    := 0;
	          #InletLineStep      := 5;
	        ELSIF (#InletLineStep=5) THEN
	          "dbTimers".Num[#i1].EE    := True;
	          "dbTimers".Num[#i1].PRE   := #TimeToReleaseInletLine;
	          IF ("dbTimers".Num[#i1].EE AND "dbTimers".Num[#i1].DN AND "dbTimers".Num[#i1].ACC>0) THEN
	            "dbTimers".Num[#i1].EE    := FALSE;
	            #InletLineStep      := 3;
	          END_IF;
	        END_IF;
	
	        IF "dbDigitalSensors".FOTOCELICA_VSTOP_DRCA_DESNO.InputF THEN // Go to filling opposite line, if line is full
	          #Mode          := 2; // Go to #CurrentStep (filing once LEVO then DESNO...)
	          #CurrentStep   := 5; // reset variables
	        END_IF;
	
	      END_IF; // #FillingLineSelector
	    // 20210506_PRA - END_IF; Check FOTOCELICA_PRED_MESTOM_LOCEVANJA only once  // "dbDigitalSensors".FOTOCELICA_PRED_MESTOM_LOCEVANJA.InputF 
	    END_REGION
	  
	    REGION MODE = 1 OUTLET HELIXS - left and right lines 
	      // *************************************************************************** //  
	      // ****************** BEGIN - Release legs from slide line ******************* // 
	      // *************************************************************************** // 
	      // LEVO
	      IF (#LeftLegIndex<=1 AND ("ph_Helix_1_DB".LeftLegIndex=2 OR #LeftFirstLegIndex<2)) THEN
	          IF "dbDigitalSensors".FOTOCELICA_LOC_IZH_DRCA_LEVO.InputF AND #LeftOutletLineStep=0  THEN
	            "dbTimers".Num[#i2].EE  := "dbMotors".VKLOP_M_TRAKA_VIJACNIKA.XS;
	            "dbTimers".Num[#i2].PRE := #TimeToReleaseOutletLine; // 200 ms
	            #LeftOutletLineStep := 1;
	          END_IF;
	          IF (#LeftOutletLineStep=1) THEN
	            "dbTimers".Num[#i2].EE  := True;
	            IF "dbDigitalSensors".FOTOCELICA_LOC_IZH_DRCA_LEVO.InputF THEN
	              "dbTimers".Num[#i2].ACC  := 0;
	            END_IF;
	            #Y7_DrcaLocev_Lev.AutoON := True;
	          END_IF;
	          IF (#LeftOutletLineStep=1) AND "dbTimers".Num[#i2].EE AND "dbTimers".Num[#i2].DN THEN
	            "dbTimers".Num[#i2].EE := False;
	            "dbTimers".Num[#i2].ACC  := 0;
	            #LeftOutletLineStep := 0;
	            #LeftLegIndex := #LeftLegIndex + 1; // Clear (#LeftLegIndex=0,  if is #LeftLegIndex=2, in phase ph_Helix_1
	            IF #LeftFirstLegIndex < 2 THEN
	              #LeftFirstLegIndex := #LeftFirstLegIndex + 1;
	            END_IF;
	          END_IF;
	      END_IF;
	  
	      // DESNO
	      IF (#RightLegIndex<=1 AND ("ph_Helix_1_DB".RightLegIndex=2 OR #RightFirstLegIndex<2)) THEN
	          IF "dbDigitalSensors".FOTOCELICA_LOC_IZH_DRCA_DESNO.InputF AND #RightOutletLineStep=0 THEN
	            "dbTimers".Num[#i3].EE  := "dbMotors".VKLOP_M_TRAKA_VIJACNIKA.XS;
	            "dbTimers".Num[#i3].PRE := #TimeToReleaseOutletLine; // 200 ms
	            #RightOutletLineStep := 1;
	          END_IF;
	          IF (#RightOutletLineStep=1) THEN
	            "dbTimers".Num[#i3].EE  := True;
	            IF "dbDigitalSensors".FOTOCELICA_LOC_IZH_DRCA_DESNO.InputF THEN
	              "dbTimers".Num[#i3].ACC  := 0;
	            END_IF;
	            #Y6_DrcaLocev_Des.AutoON := True;
	          END_IF;
	          IF (#RightOutletLineStep=1) AND "dbTimers".Num[#i3].EE AND "dbTimers".Num[#i3].DN THEN
	            "dbTimers".Num[#i3].EE := False;
	            "dbTimers".Num[#i3].ACC  := 0;
	            #RightOutletLineStep := 0;
	            #RightLegIndex := #RightLegIndex + 1; // Clear (#RightLegIndex=0,  if is #RightLegIndex=2, in phase ph_Helix_1
	            IF #RightFirstLegIndex < 2 THEN
	              #RightFirstLegIndex := #RightFirstLegIndex + 1;
	            END_IF;
	          END_IF;
	      END_IF;
	      // *************************************************************************** //  
	      // ********************* END - Release legs from slide line ****************** // 
	      // *************************************************************************** //
	    END_REGION
	
	  20:  // Fill once leg to LEVO and then once leg to DESNO, till line gets full
	    // ******************* BEGIN - ALARM STATE *********** // 
	    IF NOT #AlarmPresent THEN
	      "dbTimers".Num[#i1].FR    := False;
	      "dbTimers".Num[#i2].FR    := False;
	      "dbTimers".Num[#i3].FR    := False;
	    ELSE
	      "dbTimers".Num[#i1].FR    := True;
	      "dbTimers".Num[#i2].FR    := True;
	      "dbTimers".Num[#i3].FR    := True;
	    END_IF;
	    // ********************* END - ALARM STATE ************ // 
	
	    REGION MODE = 2 INLET HELIXS - rotation cylinder  
	    // 20210506_PRA - END_IF; Check FOTOCELICA_PRED_MESTOM_LOCEVANJA only once IF "dbDigitalSensors".FOTOCELICA_PRED_MESTOM_LOCEVANJA.InputF THEN
	      // Fill line LEVO, if leg present infront of rotation cilinder
	      IF NOT "dbDigitalSensors".FOTOCELICA_VSTOP_DRCA_LEVO.InputF AND "dbDigitalSensors".FOTOCELICA_PRED_MESTOM_LOCEVANJA.InputF AND (#InletLineStep=0) THEN
	        "dbTimers".Num[#i1].EE    := True;
	        "dbTimers".Num[#i1].PRE   := #TimeToLoadInletLine; // 10s
	        "dbTimers".Num[#i1].ACC    := 0;
	        #InletLineStep      := 1;
	      ELSIF (#InletLineStep =1) AND NOT "dbDigitalSensors".FOTOCELICA_VSTOP_DRCA_LEVO.InputF AND "dbTimers".Num[#i1].TT THEN // "dbTimers".Num[#i1].EE AND NOT "dbTimers".Num[#i1].DN 
	        "dbTimers".Num[#i1].EE    := True;  
	        #Y18_RotCilipozLevo.AutoON := True;
	      ELSIF "dbTimers".Num[#i1].EE AND "dbTimers".Num[#i1].DN AND (#InletLineStep =1) AND "dbPDO".#Y18_RotCilipozLevo THEN
	        "dbTimers".Num[#i1].ACC    := 0;
	        #InletLineStep      := 2;
	      ELSIF (#InletLineStep=2) THEN
	        "dbTimers".Num[#i1].EE    := True;
	        "dbTimers".Num[#i1].PRE   := #TimeToReleaseInletLine;
	        IF ("dbTimers".Num[#i1].EE AND "dbTimers".Num[#i1].DN AND "dbTimers".Num[#i1].ACC>0) THEN
	          #DRCA_DESNO_LATCH         := False;
	          "dbTimers".Num[#i1].ACC    := 0;
	          #InletLineStep      := 3;
	        END_IF;
	
	      // Fill line DESNO, if leg present infront of rotation cilinder
	      ELSIF NOT "dbDigitalSensors".FOTOCELICA_VSTOP_DRCA_DESNO.InputF AND "dbDigitalSensors".FOTOCELICA_PRED_MESTOM_LOCEVANJA.InputF AND (#InletLineStep=3) THEN
	        "dbTimers".Num[#i1].EE    := True;
	        "dbTimers".Num[#i1].PRE   := #TimeToLoadInletLine; // 10s
	        #InletLineStep      := 4;
	        "dbTimers".Num[#i1].ACC    := 0;
	      ELSIF (#InletLineStep =4) AND NOT "dbDigitalSensors".FOTOCELICA_VSTOP_DRCA_DESNO.InputF AND "dbTimers".Num[#i1].TT THEN // AND NOT "dbTimers".Num[#i1].DN 
	        "dbTimers".Num[#i1].EE    := True;
	        #Y17_RotCilipozDesno.AutoON := True;
	      ELSIF "dbTimers".Num[#i1].EE AND "dbTimers".Num[#i1].DN AND (#InletLineStep =4) AND "dbPDO".#Y17_RotCilipozDesno THEN
	        "dbTimers".Num[#i1].ACC    := 0;
	        #InletLineStep      := 5;
	      ELSIF (#InletLineStep=5) THEN  
	        "dbTimers".Num[#i1].EE    := True;
	        "dbTimers".Num[#i1].PRE   := #TimeToReleaseInletLine;
	        IF ("dbTimers".Num[#i1].EE AND "dbTimers".Num[#i1].DN AND "dbTimers".Num[#i1].ACC>0) THEN
	          #DRCA_LEVO_LATCH         := False;
	          "dbTimers".Num[#i1].ACC    := 0;
	          #InletLineStep      := 0;
	        END_IF;
	      END_IF;
	    // 20210506_PRA - END_IF; Check FOTOCELICA_PRED_MESTOM_LOCEVANJA only once END_IF;
	
	    IF "dbDigitalSensors".FOTOCELICA_VSTOP_DRCA_LEVO.InputF AND NOT #DRCA_LEVO_LATCH THEN // Go to filling opposite line, if line is full
	      #InletLineStep      := 3;
	      #DRCA_LEVO_LATCH    := True;
	      "dbTimers".Num[#i1].EE    := False;
	    ELSIF "dbDigitalSensors".FOTOCELICA_VSTOP_DRCA_DESNO.InputF AND NOT #DRCA_DESNO_LATCH THEN // Go to filling opposite line, if line is full
	      #InletLineStep      := 0;
	      #DRCA_DESNO_LATCH   := True;
	      "dbTimers".Num[#i1].EE    := False;
	    END_IF;
	
	    END_REGION
	  
	    REGION MODE = 2 OUTLET HELIXS - left and right lines 
	      // *************************************************************************** //  
	      // ****************** BEGIN - Release legs from slide line ******************* // 
	      // *************************************************************************** // 
	      // LEVO
	      IF (#LeftLegIndex<=1 AND ("ph_Helix_1_DB".LeftLegIndex=2 OR #LeftFirstLegIndex<2)) THEN
	          IF "dbDigitalSensors".FOTOCELICA_LOC_IZH_DRCA_LEVO.InputF AND #LeftOutletLineStep=0  THEN
	            "dbTimers".Num[#i2].EE  := "dbMotors".VKLOP_M_TRAKA_VIJACNIKA.XS;
	            "dbTimers".Num[#i2].PRE := #TimeToReleaseOutletLine; // 200 ms
	            #LeftOutletLineStep := 1;
	          END_IF;
	          IF (#LeftOutletLineStep=1) THEN
	            "dbTimers".Num[#i2].EE  := True;
	            IF "dbDigitalSensors".FOTOCELICA_LOC_IZH_DRCA_LEVO.InputF THEN
	              "dbTimers".Num[#i2].ACC  := 0;
	            END_IF;
	            #Y7_DrcaLocev_Lev.AutoON := True;
	          END_IF;
	          IF (#LeftOutletLineStep=1) AND "dbTimers".Num[#i2].EE AND "dbTimers".Num[#i2].DN THEN
	            "dbTimers".Num[#i2].EE := False;
	            "dbTimers".Num[#i2].ACC  := 0;
	            #LeftOutletLineStep := 0;
	            #LeftLegIndex := #LeftLegIndex + 1; // Clear (#LeftLegIndex=0,  if is #LeftLegIndex=2, in phase ph_Helix_1
	            IF #LeftFirstLegIndex < 2 THEN
	              #LeftFirstLegIndex := #LeftFirstLegIndex + 1;
	            END_IF;
	          END_IF;
	      END_IF;
	  
	      // DESNO
	      IF (#RightLegIndex<=1 AND ("ph_Helix_1_DB".RightLegIndex=2 OR #RightFirstLegIndex<2)) THEN
	          IF "dbDigitalSensors".FOTOCELICA_LOC_IZH_DRCA_DESNO.InputF AND #RightOutletLineStep=0 THEN
	            "dbTimers".Num[#i3].EE  := "dbMotors".VKLOP_M_TRAKA_VIJACNIKA.XS;
	            "dbTimers".Num[#i3].PRE := #TimeToReleaseOutletLine; // 200 ms
	            #RightOutletLineStep := 1;
	          END_IF;
	          IF (#RightOutletLineStep=1) THEN
	            "dbTimers".Num[#i3].EE  := True;
	            IF "dbDigitalSensors".FOTOCELICA_LOC_IZH_DRCA_DESNO.InputF THEN
	              "dbTimers".Num[#i3].ACC  := 0;
	            END_IF;
	            #Y6_DrcaLocev_Des.AutoON := True;
	          END_IF;
	          IF (#RightOutletLineStep=1) AND "dbTimers".Num[#i3].EE AND "dbTimers".Num[#i3].DN THEN
	            "dbTimers".Num[#i3].EE := False;
	            "dbTimers".Num[#i3].ACC  := 0;
	            #RightOutletLineStep := 0;
	            #RightLegIndex := #RightLegIndex + 1; // Clear (#RightLegIndex=0,  if is #RightLegIndex=2, in phase ph_Helix_1
	            IF #RightFirstLegIndex < 2 THEN
	              #RightFirstLegIndex := #RightFirstLegIndex + 1;
	            END_IF;
	          END_IF;
	      END_IF;
	      // *************************************************************************** //  
	      // ********************* END - Release legs from slide line ****************** // 
	      // *************************************************************************** //
	    END_REGION
	
	END_CASE;
	
	// ALARMS SECTION
	IF #PhaseStatus = 5 THEN
	  // Alarm 1
	  IF #Y18_RotCilipozLevo.Alarm THEN
	    "dbAlarms".PLI[#PLIIndex, 1] := 1;
	  END_IF;
	  
	  // Alarm 2
	  IF #Y17_RotCilipozDesno.Alarm THEN
	    "dbAlarms".PLI[#PLIIndex, 2] := 1;
	  END_IF;
	  
	  // Alarm 3
	  IF #Y7_DrcaLocev_Lev.Alarm THEN
	    "dbAlarms".PLI[#PLIIndex, 3] := 1;
	  END_IF;
	  
	  // Alarm 4
	  IF #Y6_DrcaLocev_Des.Alarm THEN
	    "dbAlarms".PLI[#PLIIndex, 4] := 1;
	  END_IF;
	  
	  // Alarm 5
	  // Začetna pozicija rotacijskega cilindra ni dosežena
	  IF #CurrentStep = 2 AND (#IEC_TimerOnDly_DN_1) THEN
	    "dbAlarms".PLI[#PLIIndex, 5] := 1;
	  END_IF;
	
	  // Alarms action
	  IF (NOT #AlarmPresentOLD AND #AlarmPresent) OR (NOT #InitPositionOLD AND #InitPosition) THEN
	    ; // #CurrentStep := 6;
	  END_IF;
	END_IF;
	
	#AlarmPresentOLD  := #AlarmPresent;
	#InitPositionOLD  := #InitPosition;
END_FUNCTION_BLOCK

DATA_BLOCK "op_ButtonHelix_3_DB"   // DB312
VERSION : 0.1
// stored: AutoNumber false, DBAccessibleFromOPCUA true, InstanceOfName op_ButtonHelix_3, InstanceOfType FB
"op_ButtonHelix_3"
BEGIN
   IEC_TimerOnDly_1.PT := T#0MS;
   IEC_TimerOnDly_1.IN := FALSE;
   IEC_TimerOnDly_2.PT := T#0MS;
   IEC_TimerOnDly_2.IN := FALSE;
   IEC_TimerOnDly_3.PT := T#0MS;
   IEC_TimerOnDly_3.IN := FALSE;
   IEC_TimerOnDly_4.PT := T#0MS;
   IEC_TimerOnDly_4.IN := FALSE;
   IEC_TimerOnDly_5.PT := T#0MS;
   IEC_TimerOnDly_5.IN := FALSE;
   IEC_TimerOnDly_6.PT := T#0MS;
   IEC_TimerOnDly_6.IN := FALSE;
   IEC_TimerOnDly_7.PT := T#0MS;
   IEC_TimerOnDly_7.IN := FALSE;
   IEC_TimerOnDly_8.PT := T#0MS;
   IEC_TimerOnDly_8.IN := FALSE;
   IEC_TimerOnDly_9.PT := T#0MS;
   IEC_TimerOnDly_9.IN := FALSE;
   IEC_TimerOnDly_10.PT := T#0MS;
   IEC_TimerOnDly_10.IN := FALSE;
END_DATA_BLOCK

DATA_BLOCK "ph_Helix_1_DB"   // DB310
VERSION : 0.1
// stored: AutoNumber false, DBAccessibleFromOPCUA true, InstanceOfName ph_Helix_1, InstanceOfType FB
"ph_Helix_1"
BEGIN
   IEC_TimerOnDly_1.PT := T#0MS;
   IEC_TimerOnDly_1.IN := FALSE;
   IEC_TimerOnDly_2.PT := T#0MS;
   IEC_TimerOnDly_2.IN := FALSE;
   IEC_TimerOnDly_3.PT := T#0MS;
   IEC_TimerOnDly_3.IN := FALSE;
   IEC_TimerOnDly_4.PT := T#0MS;
   IEC_TimerOnDly_4.IN := FALSE;
   IEC_TimerOnDly_5.PT := T#0MS;
   IEC_TimerOnDly_5.IN := FALSE;
   IEC_TimerOnDly_6.PT := T#0MS;
   IEC_TimerOnDly_6.IN := FALSE;
   IEC_TimerOnDly_7.PT := T#0MS;
   IEC_TimerOnDly_7.IN := FALSE;
   IEC_TimerOnDly_8.PT := T#0MS;
   IEC_TimerOnDly_8.IN := FALSE;
   IEC_TimerOnDly_9.PT := T#0MS;
   IEC_TimerOnDly_9.IN := FALSE;
   IEC_TimerOnDly_10.PT := T#0MS;
   IEC_TimerOnDly_10.IN := FALSE;
   LeftLegsArrayIndex[1..2] := TRUE;
   LeftLegsArrayIndex[3..6] := FALSE;
   RightLegsArrayIndex[1..2] := TRUE;
   RightLegsArrayIndex[3..6] := FALSE;
END_DATA_BLOCK

DATA_BLOCK "ph_LegsShifter_2_DB"   // DB311
VERSION : 0.1
// stored: AutoNumber false, DBAccessibleFromOPCUA true, InstanceOfName ph_LegsShifter_2, InstanceOfType FB
"ph_LegsShifter_2"
BEGIN
   IEC_TimerOnDly_1.PT := T#0MS;
   IEC_TimerOnDly_1.IN := FALSE;
   IEC_TimerOnDly_2.PT := T#0MS;
   IEC_TimerOnDly_2.IN := FALSE;
   IEC_TimerOnDly_3.PT := T#0MS;
   IEC_TimerOnDly_3.IN := FALSE;
   IEC_TimerOnDly_4.PT := T#0MS;
   IEC_TimerOnDly_4.IN := FALSE;
   IEC_TimerOnDly_5.PT := T#0MS;
   IEC_TimerOnDly_5.IN := FALSE;
   IEC_TimerOnDly_6.PT := T#0MS;
   IEC_TimerOnDly_6.IN := FALSE;
   IEC_TimerOnDly_7.PT := T#0MS;
   IEC_TimerOnDly_7.IN := FALSE;
   IEC_TimerOnDly_8.PT := T#0MS;
   IEC_TimerOnDly_8.IN := FALSE;
   IEC_TimerOnDly_9.PT := T#0MS;
   IEC_TimerOnDly_9.IN := FALSE;
   IEC_TimerOnDly_10.PT := T#0MS;
   IEC_TimerOnDly_10.IN := FALSE;
END_DATA_BLOCK

DATA_BLOCK "CTRL_HSC_0_DB"   // DB1
// stored: AutoNumber true, DBAccessibleFromOPCUA true, InstanceOfName CTRL_HSC, OfSystemLibElement CTRL_HSC, OfSystemLibVersion 1.0
"CTRL_HSC"
   // VAR_INPUT
   //    HSC : HW_HSC;
   //    DIR : Bool;
   //    CV : Bool;
   //    RV : Bool;
   //    PERIOD : Bool;
   //    NEW_DIR : Int;
   //    NEW_CV : DInt;
   //    NEW_RV : DInt;
   //    NEW_PERIOD : Int;
   // END_VAR
   // VAR_OUTPUT
   //    BUSY : Bool;
   //    STATUS : Word;
   // END_VAR
BEGIN
END_DATA_BLOCK

DATA_BLOCK "IEC_Timer_0_DB_OB1_1"   // DB2
{ S7_Optimized_Access := 'TRUE'; DB_Accessible_From_OPC_UA := 'FALSE' }
// stored: AutoNumber true, DBAccessibleFromOPCUA false, InstanceOfName IEC_TIMER, OfSystemLibElement IEC_TIMER, OfSystemLibVersion 1.0
"IEC_TIMER"
   // VAR
   //    PT : Time;
   //    ET { ExternalWritable := 'False'} : Time;
   //    IN : Bool;
   //    Q { ExternalWritable := 'False'} : Bool;
   // END_VAR
BEGIN
END_DATA_BLOCK
